// TIA Portal project "Buffering" (V17)

(* hardware
DEVICE "S7-1200 station_1"  S7-1200 Station
   slot 0: "Rack_0"  S7-1200 Rack  Rack  V1.0
   slot 1: "PLC_1"  CPU 1215C AC/DC/Rly  6ES7 215-1BG40-0XB0  V4.5
*)

// ===== PLC "PLC_1"  CPU 1215C AC/DC/Rly =====

VAR_GLOBAL   // PLC tag table "Default tag table"
   "Index1E" AT %MW0 : Int;
   "Index2E" AT %MW2 : Int;
   "Index1S" AT %MW4 : Int;
   "Index2S" AT %MW6 : Int;
   "CMDE_Final" AT %M10.0 : Bool;
   "CMDS_Final" AT %M10.1 : Bool;
   "X1" AT %M10.2 : Bool;
   "X2" AT %M10.3 : Bool;
   "X3" AT %M10.4 : Bool;
   "X4" AT %M10.5 : Bool;
   "X5" AT %M10.6 : Bool;
   "CMDE" AT %M10.7 : Bool;
   "CMDS" AT %M11.0 : Bool;
   "memoCMDE" AT %M11.1 : Bool;
   "memoCDMS" AT %M11.2 : Bool;
END_VAR

DATA_BLOCK "CMD"   // DB1
{ S7_Optimized_Access := 'TRUE' }
VERSION : 0.1
   VAR
      CMDE : Array[0..4] of Bool;
      CMDS : Array[0..4] of Bool;
   END_VAR
BEGIN
END_DATA_BLOCK

// folder: System blocks/Program resources

DATA_BLOCK "T3"   // DB3
{ S7_Optimized_Access := 'TRUE' }
AUTHOR : Simatic
FAMILY : IEC
NAME : IEC_TMR
VERSION : 1.0
// stored: InstanceOfName IEC_TIMER
"IEC_TIMER"
BEGIN
END_DATA_BLOCK

DATA_BLOCK "T4"   // DB4
{ S7_Optimized_Access := 'TRUE' }
AUTHOR : Simatic
FAMILY : IEC
NAME : IEC_TMR
VERSION : 1.0
// stored: InstanceOfName IEC_TIMER
"IEC_TIMER"
BEGIN
END_DATA_BLOCK

DATA_BLOCK "T5"   // DB5
{ S7_Optimized_Access := 'TRUE' }
AUTHOR : Simatic
FAMILY : IEC
NAME : IEC_TMR
VERSION : 1.0
// stored: InstanceOfName IEC_TIMER
"IEC_TIMER"
BEGIN
END_DATA_BLOCK

DATA_BLOCK "T1"   // DB6
{ S7_Optimized_Access := 'TRUE' }
AUTHOR : Simatic
FAMILY : IEC
NAME : IEC_TMR
VERSION : 1.0
// stored: InstanceOfName IEC_TIMER
"IEC_TIMER"
BEGIN
END_DATA_BLOCK

// folder: (top level)

FUNCTION "AUTO_E" : Void   // FC1, LAD
{ S7_Optimized_Access := 'TRUE' }
VERSION : 0.1
BEGIN

REGION Network 1: X1
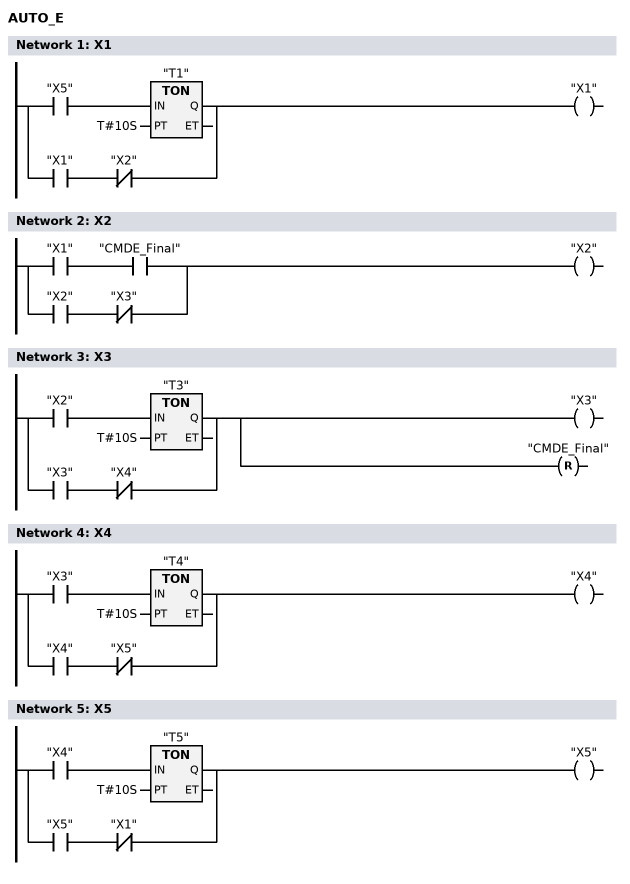
   "T1".TON(IN := "X5", PT := T#10S);
   "X1" := "T1".Q OR ("X1" AND NOT "X2");
END_REGION

REGION Network 2: X2
   RUNG wire#powerrail
      Contact( "X1" )
      Contact( "CMDE_Final" )
      wire#w1
      Coil( "X2" )
   END_RUNG
   RUNG wire#powerrail
      Contact( "X2" )
      I_Contact( "X3" )
   END_RUNG wire#w1
   // the same network as SCL:
   "X2" := ("X1" AND "CMDE_Final") OR ("X2" AND NOT "X3");
END_REGION

REGION Network 3: X3
   "T3".TON(IN := "X2", PT := T#10S);
   "X3" := "T3".Q OR ("X3" AND NOT "X4");
   IF "X3" THEN "CMDE_Final" := FALSE; END_IF;
END_REGION

REGION Network 4: X4
   "T4".TON(IN := "X3", PT := T#10S);
   "X4" := "T4".Q OR ("X4" AND NOT "X5");
END_REGION

REGION Network 5: X5
   "T5".TON(IN := "X4", PT := T#10S);
   "X5" := "T5".Q OR ("X5" AND NOT "X1");
END_REGION
END_FUNCTION

ORGANIZATION_BLOCK "Main"   // OB1, LAD, ProgramCycle
TITLE = "Main Program Sweep (Cycle)"
{ S7_Optimized_Access := 'TRUE' }
VERSION : 0.1
   VAR_TEMP   // added for the SCL form of the ladder/FBD networks
      _w1 : Bool;
   END_VAR
BEGIN

REGION Network 1
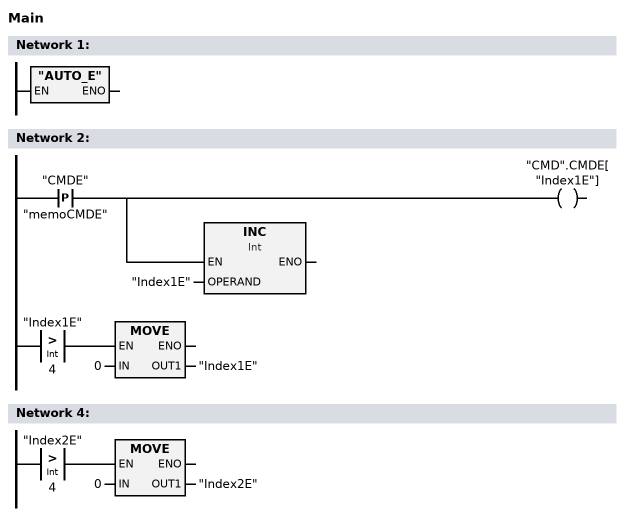
   RUNG wire#powerrail
      "AUTO_E"()
   END_RUNG
   // the same network as SCL:
   "AUTO_E"();
END_REGION

REGION Network 2
   RUNG wire#powerrail
      P_Contact(operand := "CMDE", bit := "memoCMDE")
      wire#w1
      Coil( "CMD".CMDE["Index1E"] )
   END_RUNG
   RUNG wire#w1
      { S7_Templates := "DestType := Int" } Inc( "Index1E" )
   END_RUNG
   RUNG wire#powerrail
      { S7_Templates := "SrcType := Int" } GT_Contact(in1 := "Index1E", in2 := 4)
      Move(in := 0, out1 => "Index1E")
   END_RUNG
   // the same network as SCL:
   #_w1 := "CMDE" AND NOT "memoCMDE";   // rising edge of "CMDE"
   "memoCMDE" := "CMDE";
   "CMD".CMDE["Index1E"] := #_w1;
   IF #_w1 THEN "Index1E" := "Index1E" + 1; END_IF;
   IF "Index1E" > 4 THEN "Index1E" := 0; END_IF;
END_REGION

REGION Network 3 (SCL)

   FOR "Index2E" := 0 TO 4 DO
       IF "X1" THEN
           "CMDE_Final" := "CMD".CMDE["Index2E"];
           "CMD".CMDE["Index2E"] := FALSE;
       END_IF;
   END_FOR;
END_REGION

REGION Network 4
   RUNG wire#powerrail
      { S7_Templates := "SrcType := Int" } GT_Contact(in1 := "Index2E", in2 := 4)
      Move(in := 0, out1 => "Index2E")
   END_RUNG
   // the same network as SCL:
   IF "Index2E" > 4 THEN "Index2E" := 0; END_IF;
END_REGION
END_ORGANIZATION_BLOCK